FUNCTION_BLOCK CL_AxisMCL2RightFront EXTENDS CL_AxisMC
VAR
  objAxisDriver : CL_AxisDriverL2RightFront;
END_VAR

SUPER^();

METHOD PUBLIC Init : BOOL
VAR_INPUT
  stIrrLine       : ST_LineReference;
  stAxisMotor_P	  : POINTER TO AXIS_REF;
  stAxisMaster_P  : POINTER TO AXIS_REF;
  stDriver        : POINTER TO ST_DriverAX8206_HWI;
END_VAR
Init := FALSE;
IF stDriver <> 0 THEN
  Init := objAxisDriver.Init(stDriver := stDriver);
  Init := Init AND SUPER^.InitMC(stIrrLine := stIrrLine, stAxisMotor_P := stAxisMotor_P, stAxisMaster_P := stAxisMaster_P, AxisDriver_P := ADR(objAxisDriver));
END_IF
END_METHOD

METHOD PROTECTED InitDefect : BOOL
InitDefect := SUPER^.InitDefect();
ADSLOGSTR(ADSLOG_MSGTYPE_LOG, 'CL_AxisMCL2RightFront init defect','');
END_METHOD

METHOD PROTECTED InitParams : BOOL
VAR_INPUT
END_VAR
InitParams := SUPER^.InitParams();
_sWhichAxis := 'right(L2)-front';
_lrInverse := -1.0;
END_METHOD

END_FUNCTION_BLOCK

(* stored: Version 1.1.0.1, ProductVersion 3.1.4024.12
   POU CL_AxisMCL2RightFront: Id {6a3d2686-b758-4c65-905f-34cb410c5611}, SpecialFunc None
   Method Init: Id {77f24120-24f4-4fb4-a685-b7b3cbc398cb}
   Method InitDefect: Id {a3c088b0-c881-48fa-a2f2-a087f1582cf9}
   Method InitParams: Id {ce7c670d-9ae8-438d-bcf2-f57dee39f281} *)
